(* IEC 61131-3 sources: stc/tests/ecat_fixtures, 4 files *)

(* ---- demo_bad.st ---- *)
// Deliberately broken links: one diagnostic per ECAT code.
{attribute 'qualified_only'}
VAR_GLOBAL
	// ECAT001: mistyped channel segment
	{attribute 'TcLinkTo' := 'TIID^Device 1 (EtherCAT)^DEMO.A1.00 (EK1200)^DEMO.A1.01 (EL1008)^Chanel 1^Input'}
	Typo AT %I* : BOOL;
	// ECAT002: ST_DemoEL1008 has no I9
	{attribute 'TcLinkTo' := '.I9 := TIID^Device 1 (EtherCAT)^DEMO.A1.00 (EK1200)^DEMO.A1.01 (EL1008)^Channel 8^Input'}
	NoMember : ST_DemoEL1008;
	// ECAT003: WORD on a 1-bit input
	{attribute 'TcLinkTo' := 'TIID^Device 1 (EtherCAT)^DEMO.A1.00 (EK1200)^DEMO.A1.01 (EL1008)^Channel 2^Input'}
	TooWide AT %I* : WORD;
	// ECAT004: output variable on an input entry
	{attribute 'TcLinkTo' := 'TIID^Device 1 (EtherCAT)^DEMO.A1.00 (EK1200)^DEMO.A1.01 (EL1008)^Channel 3^Input'}
	WrongDir AT %Q* : BOOL;
	// ECAT005: two variables on Channel 4
	{attribute 'TcLinkTo' := 'TIID^Device 1 (EtherCAT)^DEMO.A1.00 (EK1200)^DEMO.A1.01 (EL1008)^Channel 4^Input'}
	DupA AT %I* : BOOL;
	{attribute 'TcLinkTo' := 'TIID^Device 1 (EtherCAT)^DEMO.A1.00 (EK1200)^DEMO.A1.01 (EL1008)^Channel 4^Input'}
	DupB AT %I* : BOOL;
	// ECAT006: malformed value
	{attribute 'TcLinkTo' := '.I1 TIID^Device 1 (EtherCAT)'}
	Malformed : ST_DemoEL1008;
END_VAR

(* ---- demo_ect.st ---- *)
// Demo EtherCAT GVL: every TcLinkTo shape bound to Demo Device 1/2.
// Tests name this GVL ECT (the parser derives demo_ect from the file).
{attribute 'qualified_only'}
VAR_GLOBAL
	{attribute 'TcLinkTo' := '.I1 := TIID^Device 1 (EtherCAT)^DEMO.A1.00 (EK1200)^DEMO.A1.01 (EL1008)^Channel 1^Input;
				.I2 := TIID^Device 1 (EtherCAT)^DEMO.A1.00 (EK1200)^DEMO.A1.01 (EL1008)^Channel 2^Input;
				.I3 := TIID^Device 1 (EtherCAT)^DEMO.A1.00 (EK1200)^DEMO.A1.01 (EL1008)^Channel 3^Input;
				.I4 := TIID^Device 1 (EtherCAT)^DEMO.A1.00 (EK1200)^DEMO.A1.01 (EL1008)^Channel 4^Input;
				.I5 := TIID^Device 1 (EtherCAT)^DEMO.A1.00 (EK1200)^DEMO.A1.01 (EL1008)^Channel 5^Input;
				.I6 := TIID^Device 1 (EtherCAT)^DEMO.A1.00 (EK1200)^DEMO.A1.01 (EL1008)^Channel 6^Input;
				.I7 := TIID^Device 1 (EtherCAT)^DEMO.A1.00 (EK1200)^DEMO.A1.01 (EL1008)^Channel 7^Input;
				.I8 := TIID^Device 1 (EtherCAT)^DEMO.A1.00 (EK1200)^DEMO.A1.01 (EL1008)^Channel 8^Input;'}
	A1_01 : ST_DemoEL1008;
	{attribute 'TcLinkTo' := '.O1 := TIID^Device 1 (EtherCAT)^DEMO.A1.00 (EK1200)^DEMO.A1.02 (EL2008)^Channel 1^Output;
				.O2 := TIID^Device 1 (EtherCAT)^DEMO.A1.00 (EK1200)^DEMO.A1.02 (EL2008)^Channel 2^Output;
				.O3 := TIID^Device 1 (EtherCAT)^DEMO.A1.00 (EK1200)^DEMO.A1.02 (EL2008)^Channel 3^Output;
				.O4 := TIID^Device 1 (EtherCAT)^DEMO.A1.00 (EK1200)^DEMO.A1.02 (EL2008)^Channel 4^Output;
				.O5 := TIID^Device 1 (EtherCAT)^DEMO.A1.00 (EK1200)^DEMO.A1.02 (EL2008)^Channel 5^Output;
				.O6 := TIID^Device 1 (EtherCAT)^DEMO.A1.00 (EK1200)^DEMO.A1.02 (EL2008)^Channel 6^Output;
				.O7 := TIID^Device 1 (EtherCAT)^DEMO.A1.00 (EK1200)^DEMO.A1.02 (EL2008)^Channel 7^Output;
				.O8 := TIID^Device 1 (EtherCAT)^DEMO.A1.00 (EK1200)^DEMO.A1.02 (EL2008)^Channel 8^Output;'}
	A1_02 : ST_DemoEL2008;
	{attribute 'TcLinkTo' := '.p_stat_Enabled                 := TIID^Device 1 (EtherCAT)^DEMO.A1.00 (EK1200)^DEMO.A1.03 (EL9222-5500)^OCP Inputs Channel 1^Status^Enabled;
				.p_stat_Tripped := TIID^Device 1 (EtherCAT)^DEMO.A1.00 (EK1200)^DEMO.A1.03 (EL9222-5500)^OCP Inputs Channel 1^Status^Tripped;
				.p_Current := TIID^Device 1 (EtherCAT)^DEMO.A1.00 (EK1200)^DEMO.A1.03 (EL9222-5500)^OCP Inputs Channel 1^Current;
				.p_cmd_Reset := TIID^Device 1 (EtherCAT)^DEMO.A1.00 (EK1200)^DEMO.A1.03 (EL9222-5500)^OCP Outputs Channel 1^Control^Reset'}
	A1_03 : ST_DemoEL9222;
	{attribute 'TcLinkTo' := 'TIID^Device 1 (EtherCAT)^DEMO.A1.00 (EK1200)^DEMO.A1.04 (EL2912)^Module 3 (DEVICEIO)^FIELDVOLTAGE Field Voltage Status^Fieldvoltage Underrange'}
	A1_04_Underrange AT %I* : BOOL;
	{attribute 'TcLinkTo' := '.q_uCMD := TIID^Device 1 (EtherCAT)^DEMO.CN01.FD01 (ATV320 EtherCAT)^Outputs^CMD;
				.q_iLFR := TIID^Device 1 (EtherCAT)^DEMO.CN01.FD01 (ATV320 EtherCAT)^Outputs^LFR;
				.i_uETA := TIID^Device 1 (EtherCAT)^DEMO.CN01.FD01 (ATV320 EtherCAT)^Inputs^ETA;
				.i_iRFR := TIID^Device 1 (EtherCAT)^DEMO.CN01.FD01 (ATV320 EtherCAT)^Inputs^RFR;
				.amsaddr := TIID^Device 1 (EtherCAT)^DEMO.CN01.FD01 (ATV320 EtherCAT)^InfoData^AdsAddr;'}
	CN01 : FB_DemoDrive;
	{attribute 'TcLinkTo' := 'TIID^Device 1 (EtherCAT)^DEMO.V1 (CTEU-EtherCAT Modular)^Module 1 (VAEM-L1-S-8-PT [16DO])^Outputs^C1 Output'}
	V1_C1 AT %Q* : BYTE;
	{attribute 'TcLinkTo' := 'TIID^Device 1 (EtherCAT)^DEMO.A1.00 (EK1200)^DEMO.A1.01 (EL1008)^WcState^WcState'}
	A1_01_WcState AT %I* : BOOL;
	{attribute 'TcLinkTo' := 'TIID^Device 1 (EtherCAT)^DEMO.A1.00 (EK1200)^DEMO.A1.01 (EL1008)^InfoData^State'}
	A1_01_State AT %I* : WORD;
	{attribute 'TcLinkTo' := 'TIID^Device 1 (EtherCAT)^Inputs^DevState'}
	Dev1_DevState AT %I* : UINT;
	{attribute 'TcLinkTo' := 'TIID^Device 1 (EtherCAT)^Inputs^SlaveCount'}
	Dev1_SlaveCount AT %I* : UINT;
	{attribute 'TcLinkTo' := 'TIID^Device 1 (EtherCAT)^Inputs^Frm0State'}
	Dev1_Frm0State AT %I* : UINT;
	{attribute 'TcLinkTo' := 'TIID^Device 1 (EtherCAT)^Inputs^Frm0WcState'}
	Dev1_Frm0WcState AT %I* : UINT;
	{attribute 'TcLinkTo' := 'TIID^Device 1 (EtherCAT)^InfoData^AmsNetId'}
	Dev1_AmsNetId AT %I* : T_AmsNetIdArr;
	{attribute 'TcLinkTo' := 'TIID^Device 2 (EtherCAT)^D2.A1.01 (EL1008)^Channel 1^Input'}
	D2_I1 AT %I* : BOOL;
END_VAR

(* ---- atv320_mini.st ---- *)
// Trimmed FB_ATV320 for the CI end-to-end test (Phase 26-04). Same I/O
// names and configurator states as SVNCoreComponents FB_ATV320:
// 0 cfgWaitForPreOp, 1 cfgWriteParams, 2 cfgCommitEEPROM, 3 cfgWaitCommit,
// 4 cfgPromoteOp, 5 cfgWaitForOp, 6 cfgReady, 7 cfgErrorState.
FUNCTION_BLOCK FB_MiniATV320
VAR_INPUT
	amsaddr AT %I* : AMSADDR;
	i_xFwd : BOOL;
	i_xReset : BOOL;
	i_uETA AT %I* : UINT;
	i_iRFR AT %I* : INT;
	i_uLCR AT %I* : UINT;
	i_uDI AT %I* : UINT;
	i_eLFT AT %I* : UINT;
	i_eHMIS AT %I* : UINT;
END_VAR
VAR_OUTPUT
	q_uCMD AT %Q* : UINT;
	q_iLFR AT %Q* : INT;
	q_uOL1R AT %Q* : UINT;
	q_uACC AT %Q* : UINT;
	q_uDEC AT %Q* : UINT;
	q_xError : BOOL;
	q_xReady : BOOL;
	configState : INT;
	nLastConfigError : UDINT;
END_VAR
VAR
	sNetId : T_AmsNetId;
	nSlaveAddr : UINT;
	ecState : FB_EcGetSlaveState;
	ec : ST_EcSlaveState;
	fbSetState : FB_EcSetSlaveState;
	fbWrite : FB_EcCoESdoWrite;
	nParam : INT;
	nHSP : UINT := 500;
	nACC : UINT := 30;
	nCommitMagic : UDINT := 16#65766173;
	eta : UINT;
END_VAR
sNetId := F_CreateAmsNetId(nIds := amsaddr.netId);
nSlaveAddr := amsaddr.port;
q_uACC := 30;
q_uDEC := 30;

ecState(sNetId := sNetId, nSlaveAddr := nSlaveAddr);
IF NOT ecState.bBusy AND NOT ecState.bError THEN
	ec := ecState.state;
	ecState(bExecute := FALSE);
	ecState(bExecute := TRUE);
ELSIF ecState.bError THEN
	ecState(bExecute := FALSE);
	ecState(bExecute := TRUE);
	ec.deviceState := 0;
END_IF;

CASE configState OF
	0:
		IF ec.deviceState = 2 THEN
			configState := 1;
			nParam := 0;
		END_IF;
	1:
		CASE nParam OF
			0:
				fbWrite(sNetId := sNetId, nSlaveAddr := nSlaveAddr, nIndex := 16#2001, nSubIndex := 5,
					pSrcBuf := ADR(nHSP), cbBufLen := SIZEOF(nHSP), bExecute := TRUE);
				nParam := 1;
			1, 3:
				fbWrite();
				IF NOT fbWrite.bBusy THEN
					IF fbWrite.bError THEN
						nLastConfigError := fbWrite.nErrId;
						configState := 7;
					END_IF;
					fbWrite(bExecute := FALSE);
					nParam := nParam + 1;
				END_IF;
			2:
				fbWrite(sNetId := sNetId, nSlaveAddr := nSlaveAddr, nIndex := 16#203C, nSubIndex := 2,
					pSrcBuf := ADR(nACC), cbBufLen := SIZEOF(nACC), bExecute := TRUE);
				nParam := 3;
			4:
				configState := 2;
		END_CASE;
	2:
		fbWrite(sNetId := sNetId, nSlaveAddr := nSlaveAddr, nIndex := 16#2032, nSubIndex := 1,
			pSrcBuf := ADR(nCommitMagic), cbBufLen := SIZEOF(nCommitMagic), bExecute := TRUE);
		configState := 3;
	3:
		fbWrite();
		IF NOT fbWrite.bBusy THEN
			IF fbWrite.bError THEN
				nLastConfigError := fbWrite.nErrId;
				configState := 7;
			ELSE
				configState := 4;
			END_IF;
			fbWrite(bExecute := FALSE);
		END_IF;
	4:
		fbSetState(sNetId := sNetId, nSlaveAddr := nSlaveAddr, reqState := 16#08, bExecute := TRUE);
		configState := 5;
	5:
		fbSetState();
		IF NOT fbSetState.bBusy THEN
			IF fbSetState.bError THEN
				nLastConfigError := fbSetState.nErrId;
				configState := 7;
			ELSE
				configState := 6;
			END_IF;
			fbSetState(bExecute := FALSE);
		END_IF;
	6:
		IF ec.deviceState <> 8 THEN
			configState := 0;
		END_IF;
END_CASE;
q_xReady := configState = 6 AND ec.deviceState = 8;

// CiA402 sequencing from the decoded status word
eta := i_uETA AND 16#6F;
q_xError := (i_uETA AND 16#4F) = 16#08 OR (i_uETA AND 16#4F) = 16#0F;
IF q_xError THEN
	IF i_xReset THEN
		q_uCMD := 16#80;
	ELSE
		q_uCMD := 0;
	END_IF;
ELSIF NOT i_xFwd OR NOT q_xReady THEN
	q_uCMD := 16#06;
ELSIF eta = 16#21 THEN
	q_uCMD := 16#07;
ELSIF eta = 16#23 OR eta = 16#27 THEN
	q_uCMD := 16#0F;
ELSE
	q_uCMD := 16#06;
END_IF;
IF i_xFwd THEN
	q_iLFR := 500;
ELSE
	q_iLFR := 0;
END_IF;
END_FUNCTION_BLOCK

{attribute 'qualified_only'}
VAR_GLOBAL
	{attribute 'TcLinkTo' := '.q_uCMD := TIID^Device 3 (EtherCAT)^SIM.FD01 (ATV320 EtherCAT)^Outputs^CMD;
				.q_iLFR := TIID^Device 3 (EtherCAT)^SIM.FD01 (ATV320 EtherCAT)^Outputs^LFR;
				.q_uOL1R := TIID^Device 3 (EtherCAT)^SIM.FD01 (ATV320 EtherCAT)^Outputs^OL1R;
				.q_uACC := TIID^Device 3 (EtherCAT)^SIM.FD01 (ATV320 EtherCAT)^Outputs^ACC;
				.q_uDEC := TIID^Device 3 (EtherCAT)^SIM.FD01 (ATV320 EtherCAT)^Outputs^DEC;
				.i_uETA := TIID^Device 3 (EtherCAT)^SIM.FD01 (ATV320 EtherCAT)^Inputs^ETA;
				.i_iRFR := TIID^Device 3 (EtherCAT)^SIM.FD01 (ATV320 EtherCAT)^Inputs^RFR;
				.i_uLCR := TIID^Device 3 (EtherCAT)^SIM.FD01 (ATV320 EtherCAT)^Inputs^LCR;
				.i_uDI := TIID^Device 3 (EtherCAT)^SIM.FD01 (ATV320 EtherCAT)^Inputs^DI;
				.i_eLFT := TIID^Device 3 (EtherCAT)^SIM.FD01 (ATV320 EtherCAT)^Inputs^LFT;
				.i_eHMIS := TIID^Device 3 (EtherCAT)^SIM.FD01 (ATV320 EtherCAT)^Inputs^HMIS;
				.amsaddr := TIID^Device 3 (EtherCAT)^SIM.FD01 (ATV320 EtherCAT)^InfoData^AdsAddr;'}
	drive : FB_MiniATV320;
	{attribute 'TcLinkTo' := 'TIID^Device 3 (EtherCAT)^SIM.FD01 (ATV320 EtherCAT)^InfoData^State'}
	driveState AT %I* : UINT;
END_VAR

PROGRAM MAIN
VAR
	diagGo : BOOL;
	fbStates : FB_EcGetAllSlaveStates;
	fbMaster : FB_EcGetMasterState;
	fbCrc : FB_EcGetAllSlaveCrcErrors;
	aStates : ARRAY[0..3] OF ST_EcSlaveState;
	aCrc : ARRAY[0..3] OF UDINT;
	statesBusy, masterBusy, crcBusy : BOOL;
	masterState : WORD;
END_VAR
ECT.drive();
fbStates(sNetId := '', pStateBuf := ADR(aStates), cbBufLen := SIZEOF(aStates), bExecute := diagGo);
fbMaster(sNetId := '', bExecute := diagGo);
fbCrc(sNetId := '', pCrcErrorBuf := ADR(aCrc), cbBufLen := SIZEOF(aCrc), bExecute := diagGo);
statesBusy := fbStates.bBusy;
masterBusy := fbMaster.bBusy;
crcBusy := fbCrc.bBusy;
masterState := fbMaster.state;
END_PROGRAM

(* ---- demo_types.st ---- *)
// Types for the EtherCAT demo fixtures (Demo Device 1/2). Local stand-ins
// for AMSADDR and T_AmsNetIdArr keep the fixture self-contained.
TYPE T_AmsNetIdArr : ARRAY[0..5] OF BYTE;
END_TYPE

TYPE AMSADDR :
STRUCT
	netId : ARRAY[0..5] OF BYTE;
	port  : UINT;
END_STRUCT
END_TYPE

TYPE ST_DemoEL1008 :
STRUCT
	I1 AT %I* : BOOL;
	I2 AT %I* : BOOL;
	I3 AT %I* : BOOL;
	I4 AT %I* : BOOL;
	I5 AT %I* : BOOL;
	I6 AT %I* : BOOL;
	I7 AT %I* : BOOL;
	I8 AT %I* : BOOL;
END_STRUCT
END_TYPE

TYPE ST_DemoEL2008 :
STRUCT
	O1 AT %Q* : BOOL;
	O2 AT %Q* : BOOL;
	O3 AT %Q* : BOOL;
	O4 AT %Q* : BOOL;
	O5 AT %Q* : BOOL;
	O6 AT %Q* : BOOL;
	O7 AT %Q* : BOOL;
	O8 AT %Q* : BOOL;
END_STRUCT
END_TYPE

TYPE ST_DemoEL9222 :
STRUCT
	p_stat_Enabled AT %I* : BOOL;
	p_stat_Tripped AT %I* : BOOL;
	p_Current      AT %I* : UINT;
	p_cmd_Reset    AT %Q* : BOOL;
END_STRUCT
END_TYPE

FUNCTION_BLOCK FB_DemoDrive
VAR_OUTPUT
	uEtaSeen : UINT;
END_VAR
VAR
	q_uCMD  AT %Q* : UINT;
	q_iLFR  AT %Q* : INT;
	i_uETA  AT %I* : UINT;
	i_iRFR  AT %I* : INT;
	amsaddr AT %I* : AMSADDR;
END_VAR
uEtaSeen := i_uETA;
q_uCMD := 16#000F;
END_FUNCTION_BLOCK
